// Mitsubishi GX Works2 project: BookEX6_6 Compare   PLC: Q13UDV

// global labels: Global
VAR_GLOBAL
  bVar0 AT M5000 : BOOL;
  abArray0 AT M5010 : ARRAY [0..49] OF BOOL;
  sStr0 AT D5000 : STRING[199];
  sStr1 AT D5100 : STRING[199];
  sStr2 AT D5200 : STRING[199];
  sStr3 AT D5300 : STRING[199];
  sStr4 AT D5400 : STRING[199];
  sStr5 AT D5500 : STRING[199];
  sStr6 AT D5600 : STRING[199];
  sStr7 AT D5700 : STRING[199];
  sStr8 AT D5800 : STRING[199];
  sStr9 AT D5900 : STRING[199];
  iVar0 AT D4500 : INT;
  iVar1 AT D4501 : INT;
  iVar2 AT D4502 : INT;
  iVar3 AT D4503 : INT;
  iVar4 AT D4504 : INT;
  iVar5 AT D4505 : INT;
  iVar6 AT D4506 : INT;
  iVar7 AT D4507 : INT;
  iVar8 AT D4508 : INT;
  iVar9 AT D4509 : INT;
  dVar0 AT D4510 : DINT;
  dVar1 AT D4512 : DINT;
  dVar2 AT D4514 : DINT;
  dVar3 AT D4516 : DINT;
  dVar4 AT D4518 : DINT;
  dVar5 AT D4520 : DINT;
  dVar6 AT D4522 : DINT;
  dVar7 AT D4524 : DINT;
  dVar8 AT D4526 : DINT;
  dVar9 AT D4528 : DINT;
  wVar0 AT D4530 : WORD;
  wVar1 AT D4531 : WORD;
  wVar2 AT D4532 : WORD;
  wVar3 AT D4533 : WORD;
  wVar4 AT D4534 : WORD;
  wVar5 AT D4535 : WORD;
  wVar6 AT D4536 : WORD;
  wVar7 AT D4537 : WORD;
  wVar8 AT D4538 : WORD;
  wVar9 AT D4539 : WORD;
  dwVar0 AT D4540 : DWORD;
  dwVar1 AT D4542 : DWORD;
  dwVar2 AT D4544 : DWORD;
  dwVar3 AT D4546 : DWORD;
  dwVar4 AT D4548 : DWORD;
  dwVar5 AT D4550 : DWORD;
  dwVar6 AT D4552 : DWORD;
  dwVar7 AT D4554 : DWORD;
  dwVar8 AT D4556 : DWORD;
  dwVar9 AT D4558 : DWORD;
  fsVar0 AT D4560 : REAL;
  fsVar1 AT D4562 : REAL;
  fsVar2 AT D4564 : REAL;
  fsVar3 AT D4566 : REAL;
  fsVar4 AT D4568 : REAL;
  fsVar5 AT D4570 : REAL;
  fsVar6 AT D4572 : REAL;
  fsVar7 AT D4574 : REAL;
  fsVar8 AT D4576 : REAL;
  fsVar9 AT D4578 : REAL;
  fdVar0 AT D4580 : LREAL;
  tTime0 AT D4620 : TIME;
  tTime1 AT D4622 : TIME;
  tTime2 AT D4624 : TIME;
  tTime3 AT D4626 : TIME;
  tTime4 AT D4628 : TIME;
  tTime5 AT D4630 : TIME;
  tTime6 AT D4632 : TIME;
  tTime7 AT D4634 : TIME;
  tTime8 AT D4636 : TIME;
  tTime9 AT D4638 : TIME;
  tTime10 AT D4640 : TIME;
  bVar1 AT M5001 : BOOL;
  bVar2 AT M5002 : BOOL;
  bVar3 AT M5003 : BOOL;
  bVar4 AT M5004 : BOOL;
  bVar5 AT M5005 : BOOL;
  bVar6 AT M5006 : BOOL;
  bVar7 AT M5007 : BOOL;
  bVar8 AT M5008 : BOOL;
  bVar9 AT M5009 : BOOL;
  abArray1 AT M5060 : ARRAY [0..49] OF BOOL;
  abArray2 AT M5110 : ARRAY [0..49] OF BOOL;
  abArray3 AT M5160 : ARRAY [0..49] OF BOOL;
  abArray4 AT M5210 : ARRAY [0..49] OF BOOL;
  abArray5 AT M5260 : ARRAY [0..49] OF BOOL;
  abArray6 AT M5310 : ARRAY [0..49] OF BOOL;
  abArray7 AT M5360 : ARRAY [0..49] OF BOOL;
  abArray8 AT M5410 : ARRAY [0..49] OF BOOL;
  abArray9 AT M5460 : ARRAY [0..49] OF BOOL;
  fdVar1 AT D4584 : LREAL;
  fdVar2 AT D4588 : LREAL;
  fdVar3 AT D4592 : LREAL;
  fdVar4 AT D4596 : LREAL;
  fdVar5 AT D4600 : LREAL;
  fdVar6 AT D4604 : LREAL;
  fdVar7 AT D4608 : LREAL;
  fdVar8 AT D4612 : LREAL;
  fdVar9 AT D4616 : LREAL;
  afsPen0 AT D2000 : ARRAY [0..499] OF REAL;
  afsPen1 AT D3000 : ARRAY [0..499] OF REAL;
END_VAR
// user libraries (not included): HMI

PROGRAM ExEQ
(* structured ladder/FBD written out as ST: instructions are called as NAME(EN, inputs, outputs); _pN, _eN, _tN stand for wires *)
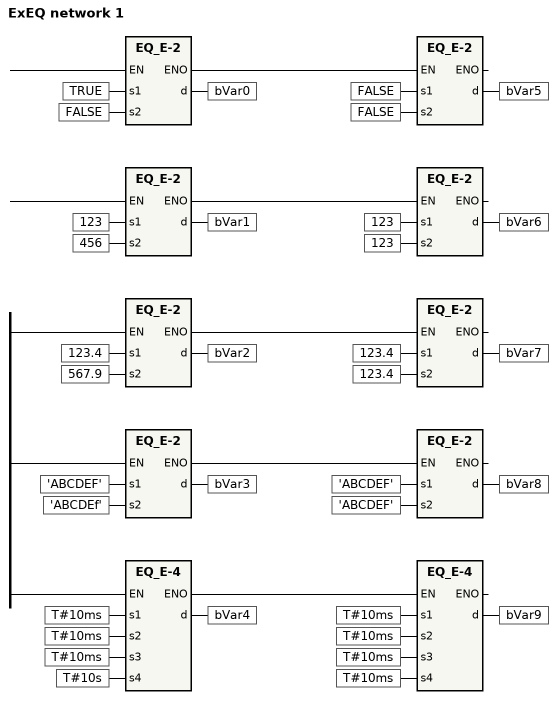
(* network 1 *)
_e1 := EQ_E(TRUE, TRUE, FALSE, bVar0);
EQ_E(_e1, FALSE, FALSE, bVar5);
_e2 := EQ_E(TRUE, 123, 456, bVar1);
EQ_E(_e2, 123, 123, bVar6);
_e3 := EQ_E(TRUE, 123.4, 567.9, bVar2);
EQ_E(_e3, 123.4, 123.4, bVar7);
_e4 := EQ_E(TRUE, 'ABCDEF', 'ABCDEf', bVar3);
EQ_E(_e4, 'ABCDEF', 'ABCDEF', bVar8);
_e5 := EQ_E(TRUE, T#10ms, T#10ms, T#10ms, T#10s, bVar4);
EQ_E(_e5, T#10ms, T#10ms, T#10ms, T#10ms, bVar9);
END_PROGRAM

PROGRAM ExGE
(* structured ladder/FBD written out as ST: instructions are called as NAME(EN, inputs, outputs); _pN, _eN, _tN stand for wires *)
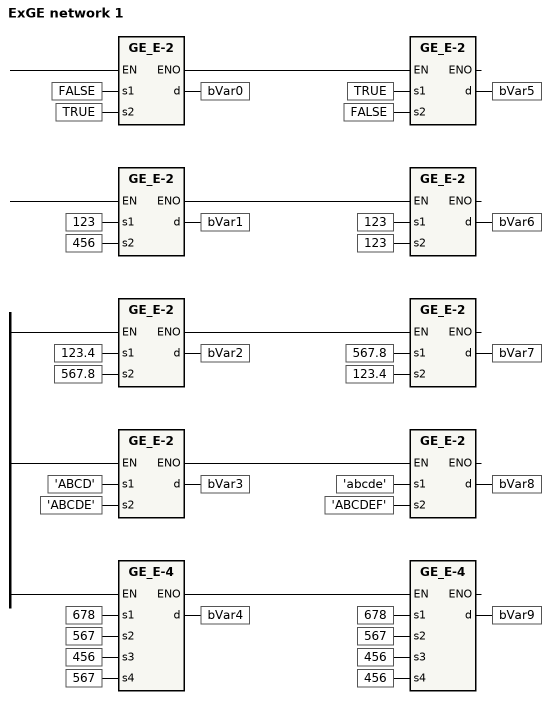
(* network 1 *)
_e1 := GE_E(TRUE, FALSE, TRUE, bVar0);
GE_E(_e1, TRUE, FALSE, bVar5);
_e2 := GE_E(TRUE, 123, 456, bVar1);
GE_E(_e2, 123, 123, bVar6);
_e3 := GE_E(TRUE, 123.4, 567.8, bVar2);
GE_E(_e3, 567.8, 123.4, bVar7);
_e4 := GE_E(TRUE, 'ABCD', 'ABCDE', bVar3);
GE_E(_e4, 'abcde', 'ABCDEF', bVar8);
_e5 := GE_E(TRUE, 678, 567, 456, 567, bVar4);
GE_E(_e5, 678, 567, 456, 456, bVar9);
END_PROGRAM

PROGRAM ExGT
(* structured ladder/FBD written out as ST: instructions are called as NAME(EN, inputs, outputs); _pN, _eN, _tN stand for wires *)
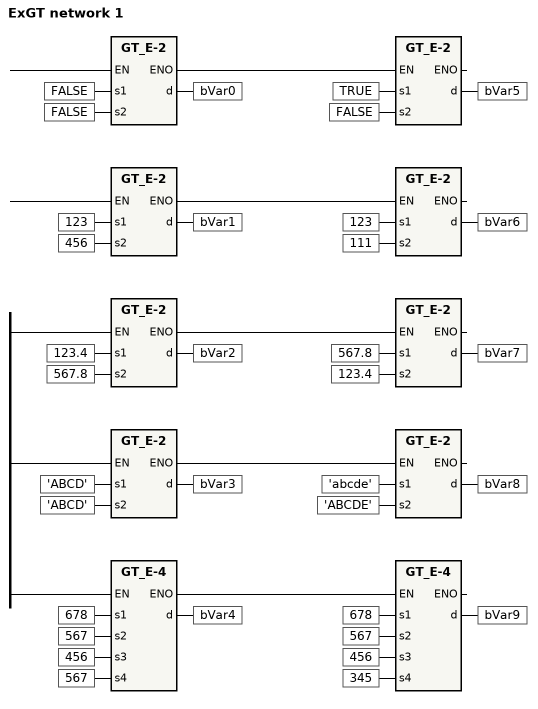
(* network 1 *)
_e1 := GT_E(TRUE, FALSE, FALSE, bVar0);
GT_E(_e1, TRUE, FALSE, bVar5);
_e2 := GT_E(TRUE, 123, 456, bVar1);
GT_E(_e2, 123, 111, bVar6);
_e3 := GT_E(TRUE, 123.4, 567.8, bVar2);
GT_E(_e3, 567.8, 123.4, bVar7);
_e4 := GT_E(TRUE, 'ABCD', 'ABCD', bVar3);
GT_E(_e4, 'abcde', 'ABCDE', bVar8);
_e5 := GT_E(TRUE, 678, 567, 456, 567, bVar4);
GT_E(_e5, 678, 567, 456, 345, bVar9);
END_PROGRAM

PROGRAM ExLE
(* structured ladder/FBD written out as ST: instructions are called as NAME(EN, inputs, outputs); _pN, _eN, _tN stand for wires *)
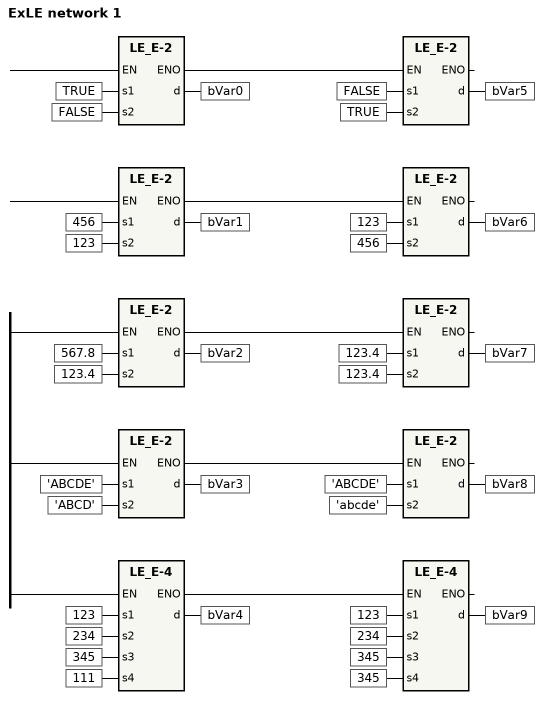
(* network 1 *)
_e1 := LE_E(TRUE, TRUE, FALSE, bVar0);
LE_E(_e1, FALSE, TRUE, bVar5);
_e2 := LE_E(TRUE, 456, 123, bVar1);
LE_E(_e2, 123, 456, bVar6);
_e3 := LE_E(TRUE, 567.8, 123.4, bVar2);
LE_E(_e3, 123.4, 123.4, bVar7);
_e4 := LE_E(TRUE, 'ABCDE', 'ABCD', bVar3);
LE_E(_e4, 'ABCDE', 'abcde', bVar8);
_e5 := LE_E(TRUE, 123, 234, 345, 111, bVar4);
LE_E(_e5, 123, 234, 345, 345, bVar9);
END_PROGRAM

PROGRAM ExLT
(* structured ladder/FBD written out as ST: instructions are called as NAME(EN, inputs, outputs); _pN, _eN, _tN stand for wires *)
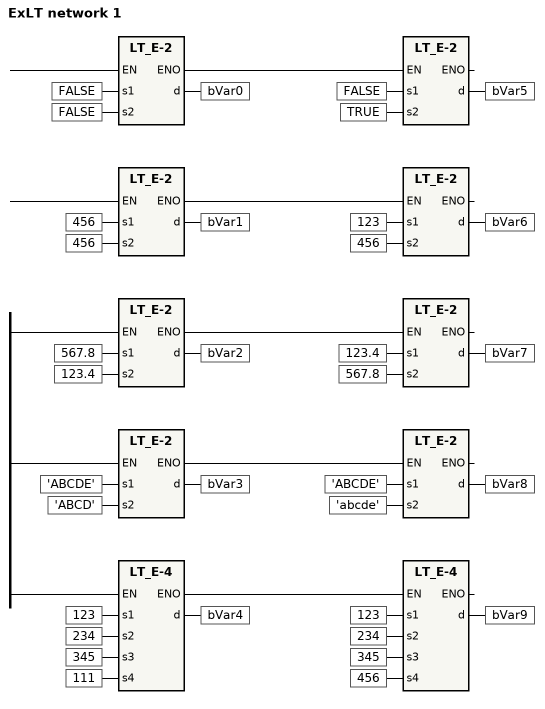
(* network 1 *)
_e1 := LT_E(TRUE, FALSE, FALSE, bVar0);
LT_E(_e1, FALSE, TRUE, bVar5);
_e2 := LT_E(TRUE, 456, 456, bVar1);
LT_E(_e2, 123, 456, bVar6);
_e3 := LT_E(TRUE, 567.8, 123.4, bVar2);
LT_E(_e3, 123.4, 567.8, bVar7);
_e4 := LT_E(TRUE, 'ABCDE', 'ABCD', bVar3);
LT_E(_e4, 'ABCDE', 'abcde', bVar8);
_e5 := LT_E(TRUE, 123, 234, 345, 111, bVar4);
LT_E(_e5, 123, 234, 345, 456, bVar9);
END_PROGRAM

PROGRAM ExMin_Max
VAR
  Min_Max_1 : Min_Max;
END_VAR
(* structured ladder/FBD written out as ST: instructions are called as NAME(EN, inputs, outputs); _pN, _eN, _tN stand for wires *)
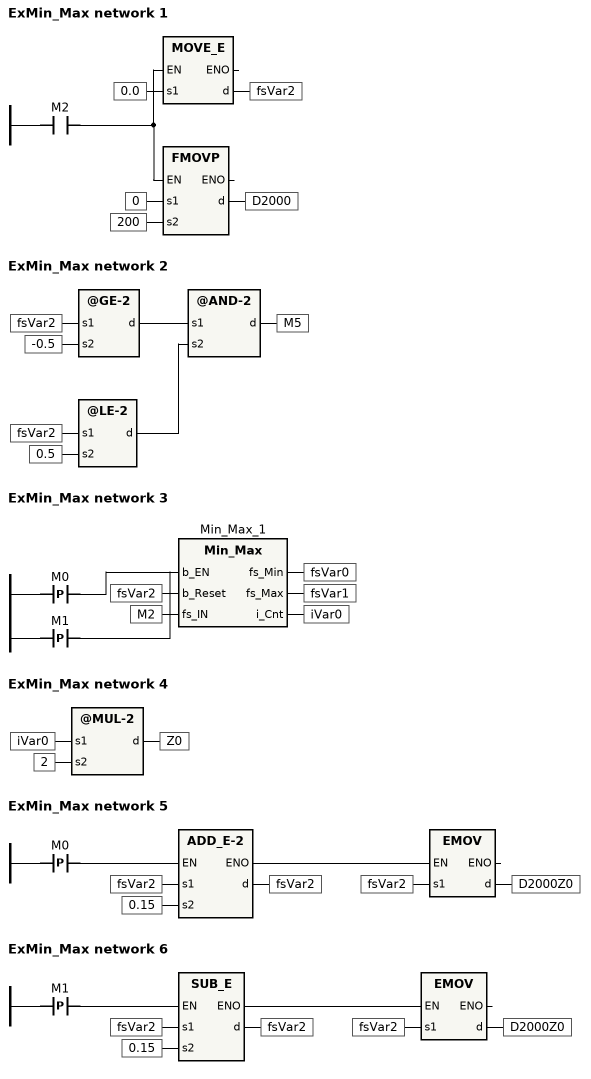
(* network 1 *)
MOVE_E(M2, 0.0, fsVar2);
FMOVP(M2, 0, 200, D2000);
(* network 2 *)
M5 := @AND-2(@GE-2(fsVar2, -0.5), @LE-2(fsVar2, 0.5));
(* network 3 *)
Min_Max_1(b_EN := LDP(TRUE, M0) OR LDP(TRUE, M1), b_Reset := fsVar2, fs_IN := M2, fs_Min => fsVar0, fs_Max => fsVar1, i_Cnt => iVar0);
(* network 4 *)
Z0 := @MUL-2(iVar0, 2);
(* network 5 *)
_e1 := ADD_E(LDP(TRUE, M0), fsVar2, 0.15, fsVar2);
EMOV(_e1, fsVar2, D2000Z0);
(* network 6 *)
_e1 := SUB_E(LDP(TRUE, M1), fsVar2, 0.15, fsVar2);
EMOV(_e1, fsVar2, D2000Z0);
END_PROGRAM

PROGRAM ExNE
(* structured ladder/FBD written out as ST: instructions are called as NAME(EN, inputs, outputs); _pN, _eN, _tN stand for wires *)
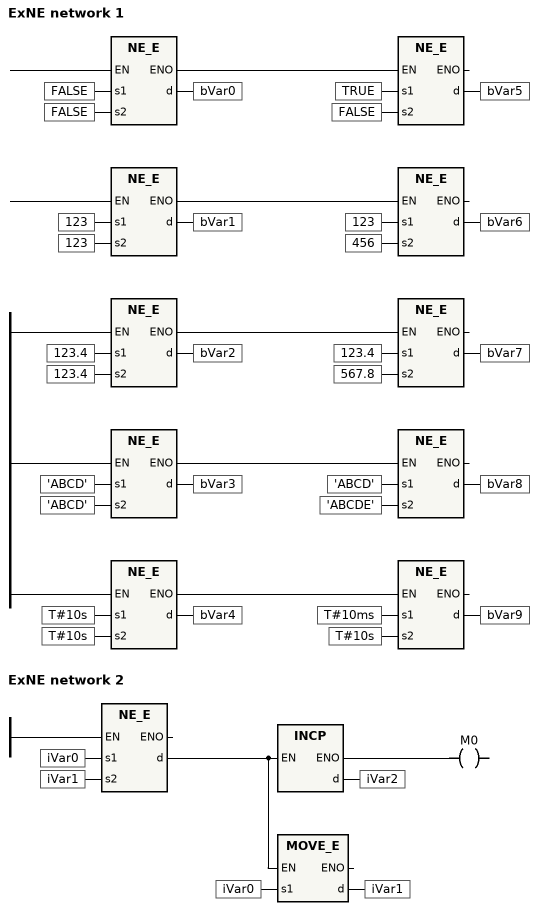
(* network 1 *)
_e1 := NE_E(TRUE, FALSE, FALSE, bVar0);
NE_E(_e1, TRUE, FALSE, bVar5);
_e2 := NE_E(TRUE, 123, 123, bVar1);
NE_E(_e2, 123, 456, bVar6);
_e3 := NE_E(TRUE, 123.4, 123.4, bVar2);
NE_E(_e3, 123.4, 567.8, bVar7);
_e4 := NE_E(TRUE, 'ABCD', 'ABCD', bVar3);
NE_E(_e4, 'ABCD', 'ABCDE', bVar8);
_e5 := NE_E(TRUE, T#10s, T#10s, bVar4);
NE_E(_e5, T#10ms, T#10s, bVar9);
(* network 2 *)
NE_E(TRUE, iVar0, iVar1, _t1);
_e2 := INCP(_t1, iVar2);
M0 := _e2;
MOVE_E(_t1, iVar0, iVar1);
END_PROGRAM

PROGRAM ExSchmitt
VAR
  fbSchmitt : Schmitt;
  ix : INT;
END_VAR
;

IF M2 THEN (* STOP *)
	M0 := FALSE;
	M1 := FALSE;
	iVar0 := 0;
	fsVar0 := 0.0;
	fsVar8 := 1.0;
	fsVar9 := -1.0;
	FOR ix := 0 TO 359 DO 
		afsPen0[ix] := 0.0;
	END_FOR;
	RETURN;
END_IF;

IF M0 THEN (* Up *)
	IF fsVar0 < 0.5 THEN
		fsVar0 := fsVar0 + 0.07;
	ELSE
		fsVar0 := fsVar0 + 0.03;
	END_IF;
	IF fsVar0 > 1.0 THEN 
		fsVar0 := 1.0;
	END_IF;
END_IF;

IF M1 THEN (* Dw *)
	IF fsVar0 < 0.5 THEN
		fsVar0 := fsVar0 - 0.07;
	ELSE
		fsVar0 := fsVar0 - 0.03;
	END_IF;
	IF fsVar0 < 0.0 THEN 
		fsVar0 := 0.0;
	END_IF;
END_IF;
afsPen0[iVar0] := fsVar0;
iVar0 := iVar0 +1;
IF iVar0 > 359 THEN
	iVar0 := 359;
	FOR ix := 1 TO 359 DO 
		afsPen0[ix-1] := afsPen0[ix];
	END_FOR;
END_IF;

fbSchmitt(fs_IN := fsVar0, fs_High := 0.8, fs_Low := 0.6);
M5 := fbSchmitt.b_Q;
M6 := fbSchmitt.b_Win;

IF NOT M5 THEN 
	M0 := FALSE;
	M1 := TRUE;
ELSE
	M0 := TRUE;
	M1 := FALSE;	
END_IF;
END_PROGRAM

PROGRAM ExWindow
(* structured ladder/FBD written out as ST: instructions are called as NAME(EN, inputs, outputs); _pN, _eN, _tN stand for wires *)
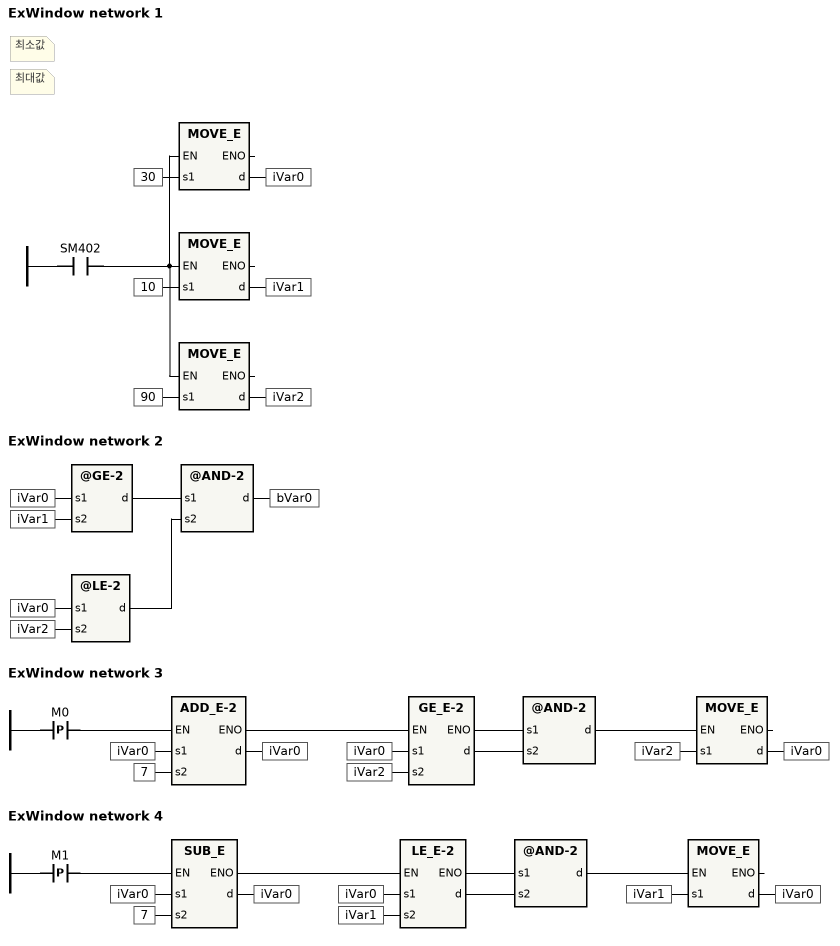
(* network 1 *)
(* 최소값 *)
(* 최대값 *)
MOVE_E(SM402, 30, iVar0);
MOVE_E(SM402, 10, iVar1);
MOVE_E(SM402, 90, iVar2);
(* network 2 *)
bVar0 := @AND-2(@GE-2(iVar0, iVar1), @LE-2(iVar0, iVar2));
(* network 3 *)
_e1 := ADD_E(LDP(TRUE, M0), iVar0, 7, iVar0);
_e3 := GE_E(_e1, iVar0, iVar2, _t2);
MOVE_E(@AND-2(_e3, _t2), iVar2, iVar0);
(* network 4 *)
_e1 := SUB_E(LDP(TRUE, M1), iVar0, 7, iVar0);
_e3 := LE_E(_e1, iVar0, iVar1, _t2);
MOVE_E(@AND-2(_e3, _t2), iVar1, iVar0);
END_PROGRAM

FUNCTION_BLOCK DispHMI1
VAR_INPUT
  b_RST : BOOL;
  b_WR : BOOL;
  dw_Data : DWORD;
  b_Data : BOOL;
END_VAR
VAR
  Buffer : ARRAY [0..7] OF WordBit;
  ix : INT;
END_VAR
;
IF LDP(TRUE, b_RST) OR  LDP(TRUE, b_WR) THEN
	IF LDP(TRUE, b_RST) THEN
		FOR ix := 0 TO 7 BY 1 DO
			Buffer[ix].Data := 0;
			Buffer[ix].Flag := FALSE;
		END_FOR;
	ELSE
		FOR ix := 0 TO 6 BY 1 DO
			Buffer[7-ix].Data := Buffer[6-ix].Data; 
			Buffer[7-ix].Flag := Buffer[6-ix].Flag;
		END_FOR;
		Buffer[0].Data := dw_Data;
		Buffer[0].Flag := b_Data;
 	END_IF;
 	FOR ix := 0 TO 7 BY 1 DO
		adwD10[ix] := Buffer[ix].Data; 
		abM10[ix] := Buffer[ix].Flag;
	END_FOR;
END_IF;
END_FUNCTION_BLOCK

FUNCTION_BLOCK DispHMI2
VAR_INPUT
  Str0 : STRING[199];
  Str1 : STRING[199];
  Str2 : STRING[199];
  Str3 : STRING[199];
  Str4 : STRING[199];
  Str5 : STRING[199];
  Str6 : STRING[199];
  Str7 : STRING[199];
  Str8 : STRING[199];
  Str9 : STRING[199];
END_VAR
(* structured ladder/FBD written out as ST: instructions are called as NAME(EN, inputs, outputs); _pN, _eN, _tN stand for wires *)
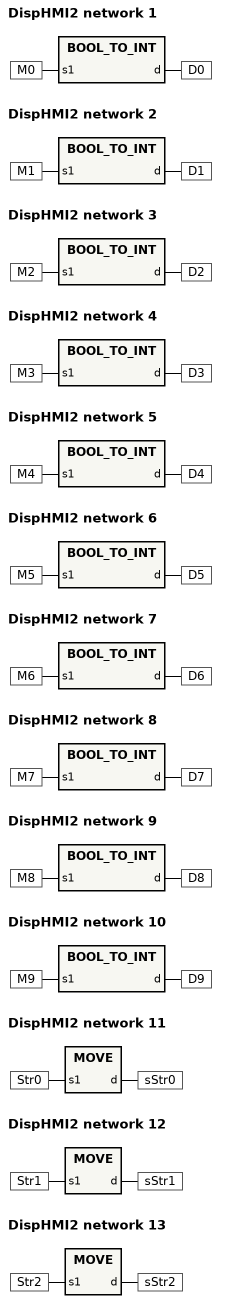
(* network 1 *)
D0 := BOOL_TO_INT(M0);
(* network 2 *)
D1 := BOOL_TO_INT(M1);
(* network 3 *)
D2 := BOOL_TO_INT(M2);
(* network 4 *)
D3 := BOOL_TO_INT(M3);
(* network 5 *)
D4 := BOOL_TO_INT(M4);
(* network 6 *)
D5 := BOOL_TO_INT(M5);
(* network 7 *)
D6 := BOOL_TO_INT(M6);
(* network 8 *)
D7 := BOOL_TO_INT(M7);
(* network 9 *)
D8 := BOOL_TO_INT(M8);
(* network 10 *)
D9 := BOOL_TO_INT(M9);
(* network 11 *)
sStr0 := MOVE(Str0);
(* network 12 *)
sStr1 := MOVE(Str1);
(* network 13 *)
sStr2 := MOVE(Str2);
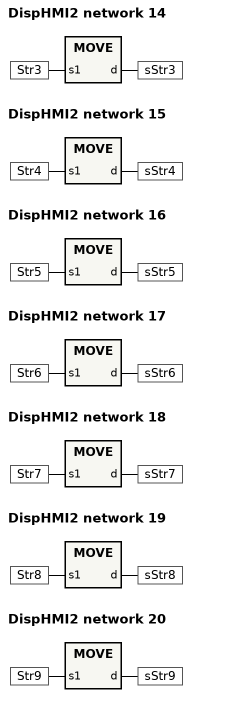
(* network 14 *)
sStr3 := MOVE(Str3);
(* network 15 *)
sStr4 := MOVE(Str4);
(* network 16 *)
sStr5 := MOVE(Str5);
(* network 17 *)
sStr6 := MOVE(Str6);
(* network 18 *)
sStr7 := MOVE(Str7);
(* network 19 *)
sStr8 := MOVE(Str8);
(* network 20 *)
sStr9 := MOVE(Str9);
END_FUNCTION_BLOCK

FUNCTION_BLOCK Min_Max
VAR_INPUT
  b_EN : BOOL;
  b_Reset : BOOL;
END_VAR
VAR_OUTPUT
  fs_Min : REAL;
  fs_Max : REAL;
  i_Cnt : INT;
END_VAR
VAR_INPUT
  fs_IN : REAL;
END_VAR
;
IF b_Reset THEN
	fs_Min := fs_IN;
	fs_Max := fs_IN;
	i_Cnt := 0;
ELSIF b_EN THEN
	i_Cnt := i_Cnt+1;
	IF fs_IN < fs_Min THEN fs_Min := fs_IN;  
	ELSIF fs_IN > fs_Max THEN fs_Max := fs_IN;  
	END_IF;
END_IF;
END_FUNCTION_BLOCK

FUNCTION_BLOCK Schmitt
VAR_INPUT
  fs_IN : REAL;
  fs_High : REAL;
  fs_Low : REAL;
END_VAR
VAR_OUTPUT
  b_Q : BOOL;
  b_Win : BOOL;
END_VAR
;
IF fs_IN < fs_Low THEN
	b_Q := TRUE;
	b_Win := FALSE;
ELSIF fs_IN > fs_High THEN
	b_Q := FALSE;
	b_Win := FALSE;
ELSE
	b_Win := TRUE;
END_IF;
END_FUNCTION_BLOCK
